FUNCTION_BLOCK FB_CylinderAlternative EXTENDS fbComponent IMPLEMENTS ITF_CylinderAlternative
VAR_INPUT
	(*~
		<docu>
			<summary>
				Home position sensor.
			</summary>	
		</docu>
	~*)
	{attribute wpf [Container(Layout.UniformGrid)]}
	{attribute wpf [Group(Layout.GroupBox, "Inputs")]}	
	{attribute addProperty Name "Home position sensor"}
	_atHomePos : BOOL;
	(*~
		<docu>
			<summary>
				Working position sensor.
			</summary>	
		</docu>
	~*) 
	{attribute addProperty Name "Work position sensor"}
	_atWorkPos : BOOL; 
END_VAR
VAR_OUTPUT
	(*~
		<docu>
			<summary>
				Move to working home position signal.
			</summary>	
		</docu>
	~*)
	{attribute wpf [Container(Layout.UniformGrid)]}
	{attribute wpf [Group(Layout.GroupBox, "Outputs")]}	
	{attribute addProperty Name "Move to home position actuator"}
	toHomePos : BOOL;
	(*~
		<docu>
			<summary>
				Move to working posistion signal.
			</summary>	
		</docu>
	~*)
	{attribute addProperty Name "Move to work position actuator"}
	toWorkPos : BOOL;
END_VAR

VAR
	{attribute wpf [Container(Layout.UniformGrid)]}
	{attribute wpf [Group(Layout.GroupBox, "Manual controls")]}
	{attribute addProperty Name "Manual move to work position"}
	_manualMoveToWork : BOOL;
	{attribute addProperty Name "Manual move to home position"}
	_manualMoveToHome : BOOL;
END_VAR

{attribute 'TcRpcEnable'}
METHOD INTERNAL _MoveToHomeTest : BOOL
_MoveToHomeTest := MoveToHome();
_atHomePos := TRUE;
_atWorkPos := FALSE;
END_METHOD

{attribute 'TcRpcEnable'}
METHOD INTERNAL _MoveToWorkTest : BOOL
_MoveToWorkTest := MoveToWork();
_atHomePos := FALSE;
_atWorkPos := TRUE;
END_METHOD

PROPERTY AtHome : bool
GET
AtHome := _atHomePos;
END_GET
END_PROPERTY

PROPERTY AtWork : bool
GET
AtWork := _atWorkPos;
END_GET
END_PROPERTY

METHOD PROTECTED  ManualControl
IF(_manualMoveToWork) AND_THEN THIS^.MoveToWork() THEN _manualMoveToWork := FALSE; END_IF
IF(_manualMoveToHome) AND_THEN THIS^.MoveToHome() THEN _manualMoveToHome := FALSE; END_IF
END_METHOD

(*~
	<docu>
		<summary>
			Moves the piston into home position.
		</summary>
		<returns>True when home position sensor is reached.</returns>
	</docu>
~*)
METHOD MoveToHome : BOOL
toHomePos := TRUE;
toWorkPos := FALSE; 
MoveToHome := _atHomePos;
Info('Moving home');
END_METHOD

(*~
	<docu>
		<summary>
			Moves the piston into working position.
		</summary>
		<returns>True when working position sensor is reached.</returns>
	</docu>
~*)
METHOD MoveToWork : BOOL
toWorkPos := TRUE; 
toHomePos := FALSE;
MoveToWork := _atWorkPos;
Info('Moving to work');
END_METHOD

PROPERTY MovingToHomePosition : BOOL
GET
MovingToHomePosition := toHomePos AND NOT AtHome;
END_GET
END_PROPERTY

PROPERTY MovingToWorkPosition : BOOL
GET
MovingToWorkPosition := toWorkPos AND NOT AtWork;
END_GET
END_PROPERTY

END_FUNCTION_BLOCK

(* stored: Version 1.1.0.1, ProductVersion 3.1.4024.4
   POU FB_CylinderAlternative: Id {fe4e2550-76ec-4019-82bb-e68b2cbe4d49}, SpecialFunc None
   Folder _tests: Id {2cbd4d6b-2a4a-49b8-b437-ed7c5a45b843}
   Method _MoveToHomeTest: Id {9ef39d14-16a3-4bc8-b330-33d879f1f7f9}
   Method _MoveToWorkTest: Id {7ebcdca4-683e-48c8-8052-33f48bfaaa19}
   Property AtHome: Id {d06903a0-9230-4f9a-9ffc-ed1726b8d4b9}
   Get Get: Id {2309dcb2-6c63-44cf-85e0-e6e2754836eb}
   Property AtWork: Id {c484892b-8ab6-4a33-a377-7a200a12d81a}
   Get Get: Id {b963dd74-98d0-4492-a086-b714bde49f51}
   Method ManualControl: Id {94b70f4e-af12-4cab-8a9f-9a3da438ebd4}
   Method MoveToHome: Id {40560f4f-3063-47a8-8b62-1f2968f73b89}
   Method MoveToWork: Id {d11735f5-ce5f-4a7f-8109-144749721e33}
   Property MovingToHomePosition: Id {c94ca31b-f1a7-4e9c-924a-99c283b9e845}
   Get Get: Id {d3fba5fc-adab-4ae3-98d6-53a9febdae02}
   Property MovingToWorkPosition: Id {d72e3e24-913b-428d-b64e-1186d58c9b4e}
   Get Get: Id {e36869bb-201c-4364-9d52-ab9f51852e16} *)
